{attribute 'no_explicit_call' := 'do not call this function block directly'} 
FUNCTION_BLOCK AutomationEngineAdsLogger EXTENDS TwinCAT_OpenFramework_Core.Object
VAR
	_ClassName : STRING := __POUNAME();
	
	_AutomationEngine : REFERENCE TO AutomationEngine;

	_DeferredLoggingRecords : TwinCAT_OpenFramework_Collections.PointerList(POINTER_TYPE.OBJECT_POINTER); // of POINTER TO DeferredLoggingRecord
	_LastMessage : ERROR_MESSAGE;
END_VAR

{attribute 'monitoring' := 'call'}
PROPERTY ClassName : STRING
GET
ClassName := _ClassName;
END_GET
END_PROPERTY

METHOD Execute : BOOL
VAR_INPUT
	codeExecutionPhase : BOOL;
END_VAR
VAR
	_Record : POINTER TO DeferredLoggingRecord;
END_VAR
WHILE _DeferredLoggingRecords.Count > 0 DO
	_Record := _DeferredLoggingRecords.Get(0);

	IF codeExecutionPhase THEN
		LogMessage(_Record^.Level, WideStringHelper.ConcatStrings255("~", _Record^.Message));		
	END_IF
		
	_DeferredLoggingRecords.RemoveAt(0, TRUE);
END_WHILE
END_METHOD

METHOD FB_exit : BOOL
VAR_INPUT
	bInCopyCode : BOOL; // if TRUE, the exit method is called for exiting an instance that is copied afterwards (online change).
END_VAR
_DeferredLoggingRecords.Clear(TRUE);
END_METHOD

METHOD FB_init : BOOL
VAR_INPUT
	(* if TRUE, the retain variables are initialized (warm start / cold start)*)
	bInitRetains	: BOOL;
	(* if TRUE, the instance afterwards gets moved into the copy code (online change)*)
	bInCopyCode	: BOOL;
	automationEngine : REFERENCE TO AutomationEngine;
END_VAR
_AutomationEngine REF= automationEngine;
END_METHOD

METHOD LogException
VAR_INPUT
	exception : REFERENCE TO Exception;
END_VAR
IF NOT __ISVALIDREF(exception) THEN
	RETURN;
END_IF

IF exception.Fatal THEN
	LogMessage(LOGGING_LEVEL.FATAL_ERROR, exception.GetMessage(TRUE, TRUE));
ELSE
	LogMessage(LOGGING_LEVEL.ERROR, exception.GetMessage(TRUE, TRUE));
END_IF
END_METHOD

METHOD LogMessage
VAR_INPUT
	level : LOGGING_LEVEL;	
	message : ERROR_MESSAGE;
END_VAR
VAR
	loggingRecord : POINTER TO DeferredLoggingRecord;
END_VAR
IF _AutomationEngine.CodeExecutionPhase THEN
	// check for message flood
	IF _LastMessage = message THEN
		RETURN;
	END_IF

	CASE level OF
		LOGGING_LEVEL.INFORMATION:
			IF level >= LoggingSettings.MinLoggingLevel THEN
				Tc2_System.ADSLOGSTR(ADSLOG_MSGTYPE_HINT AND ADSLOG_MSGTYPE_LOG, WSTRING_TO_STRING(message), '');					
			END_IF
			
		LOGGING_LEVEL.WARNING:
			IF level >= LoggingSettings.MinLoggingLevel THEN
				Tc2_System.ADSLOGSTR(ADSLOG_MSGTYPE_WARN AND ADSLOG_MSGTYPE_LOG, WSTRING_TO_STRING(message), '');					
			END_IF
			
		LOGGING_LEVEL.ERROR:
			IF level >= LoggingSettings.MinLoggingLevel THEN
				Tc2_System.ADSLOGSTR(ADSLOG_MSGTYPE_ERROR AND ADSLOG_MSGTYPE_LOG, WSTRING_TO_STRING(message), '');
			END_IF

		LOGGING_LEVEL.FATAL_ERROR:
			Tc2_System.ADSLOGSTR(ADSLOG_MSGTYPE_ERROR AND ADSLOG_MSGTYPE_LOG, WSTRING_TO_STRING(message), '');
	END_CASE
	
	_LastMessage := message;
ELSE
	// prevent memory leaking
	IF _DeferredLoggingRecords.Count < 100 THEN
		loggingRecord := __NEW(DeferredLoggingRecord);
		
		loggingRecord^.Level := level;
		loggingRecord^.Message := message;
		
		_DeferredLoggingRecords.Append(loggingRecord);		
	END_IF
END_IF
END_METHOD

{attribute 'monitoring' := 'call'}
PROPERTY Size : ULINT
GET
Size := XSIZEOF(THIS^);
END_GET
END_PROPERTY

END_FUNCTION_BLOCK

(* stored: Version 1.1.0.1
   POU AutomationEngineAdsLogger: Id {8a52fac2-0a5d-426b-84b1-4be3d24ef859}, SpecialFunc None
   Property ClassName: Id {a303aabd-1131-4065-8bf6-69d62a2ea9a2}
   Get Get: Id {8fa6fd96-da3c-4d4f-9036-392ae9e00cc9}
   Method Execute: Id {4ca73342-3129-4db1-bfe8-ce9f31717da5}
   Method FB_exit: Id {65b9e85b-cb70-4901-bf73-3fd94ecc6145}
   Method FB_init: Id {20b723fe-fcfc-43ed-88ec-de7d067f4fc1}
   Method LogException: Id {faf433b2-0e52-4cd4-a411-728b0125685c}
   Method LogMessage: Id {0709925d-8c1e-4a16-8695-6c58268bf6fc}
   Property Size: Id {695541b8-e73b-4c08-b887-91a6e80a6878}
   Get Get: Id {85961c4e-4a8a-487a-a478-61fc48b9a371} *)
